(* Logix 5000 project; controller SX_V040001_C001 vendor 1 type 14 code 77 rev 16.23; software revision 16.04; part 7 of 35 *)
(* tags used below, declared in another part *)
   ALARM_BITS : INT[10];
   ALL_KINDS : INT[90];
   average_current : DINT;
   Basic : INT;
   DRIVE : INT[32];
   EMPTYING : INT[18];
   FP_ALARM_EXIST : BOOL;
   G_AInput : DINT[8];
   G_DInput : DINT[3];
   G_DOutput : DINT[3];
   loading : INT[19];
   m_alarm_exist : BOOL;
   m_alarm_horn : BOOL;
   m_notstop : BOOL;
   M_VKE_1 : BOOL;
   METERING : INT[44];
   PARAMETER : INT[501];
   pointer_dump_current : DINT;
   T_MET12_END : TIMER;
   T_MET13_END : TIMER;
   T_MET14_END : TIMER;
   T_MET_VALVE_13 : TIMER;
   T_MET_VALVE_14 : TIMER;
(* MainProgram, continued *)

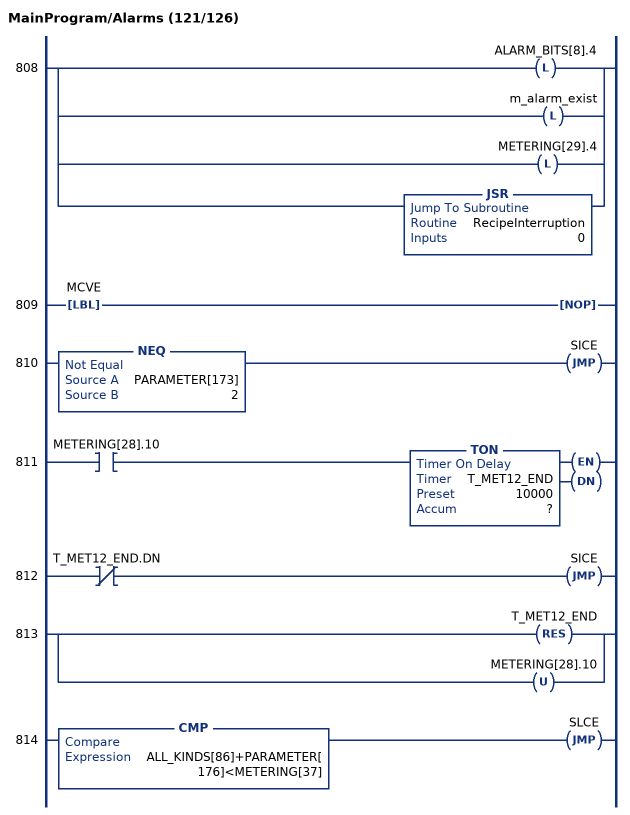
   [picture p142: MainProgram/Alarms rungs 808-814]
   808: [OTL(ALARM_BITS[8].4) ,OTL(m_alarm_exist) ,OTL(METERING[29].4) ,JSR(RecipeInterruption,0) ];
   809: LBL(MCVE)NOP();
   810: NEQ(PARAMETER[173],2)JMP(SICE);
   811: XIC(METERING[28].10)TON(T_MET12_END,?,?);
   812: XIO(T_MET12_END.DN)JMP(SICE);
   813: [RES(T_MET12_END) ,OTU(METERING[28].10) ];
   814: CMP(ALL_KINDS[86]+PARAMETER[176]<METERING[37])JMP(SLCE);
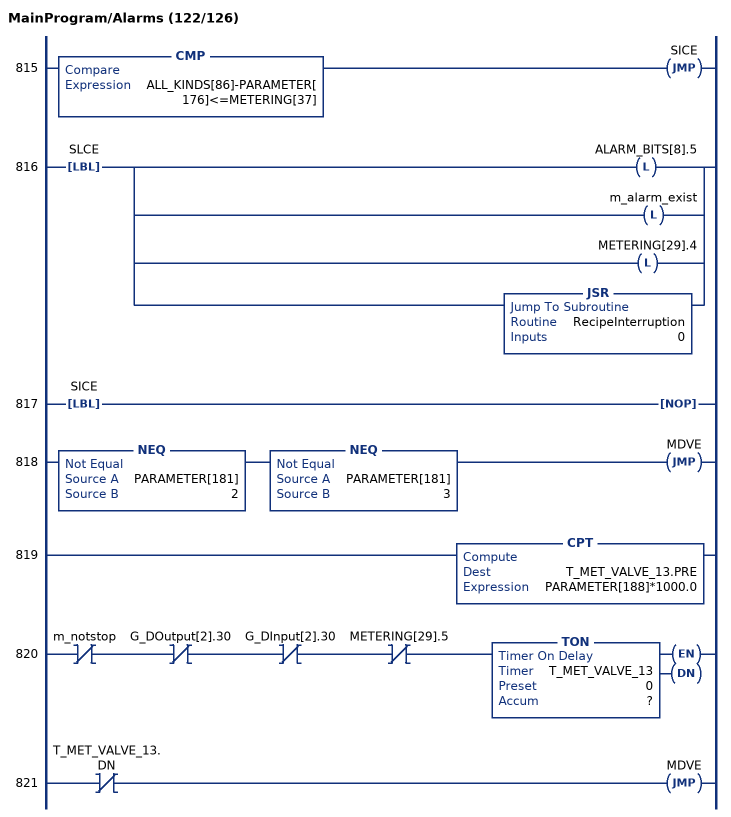
   815: CMP(ALL_KINDS[86]-PARAMETER[176]<=METERING[37])JMP(SICE);
   816: LBL(SLCE)[OTL(ALARM_BITS[8].5) ,OTL(m_alarm_exist) ,OTL(METERING[29].4) ,JSR(RecipeInterruption,0) ];
   817: LBL(SICE)NOP();
   818: NEQ(PARAMETER[181],2)NEQ(PARAMETER[181],3)JMP(MDVE);
   819: CPT(T_MET_VALVE_13.PRE,PARAMETER[188]*1000.0);
   820: XIO(m_notstop)XIO(G_DOutput[2].30)XIO(G_DInput[2].30)XIO(METERING[29].5)TON(T_MET_VALVE_13,?,?);
   821: XIO(T_MET_VALVE_13.DN)JMP(MDVE);
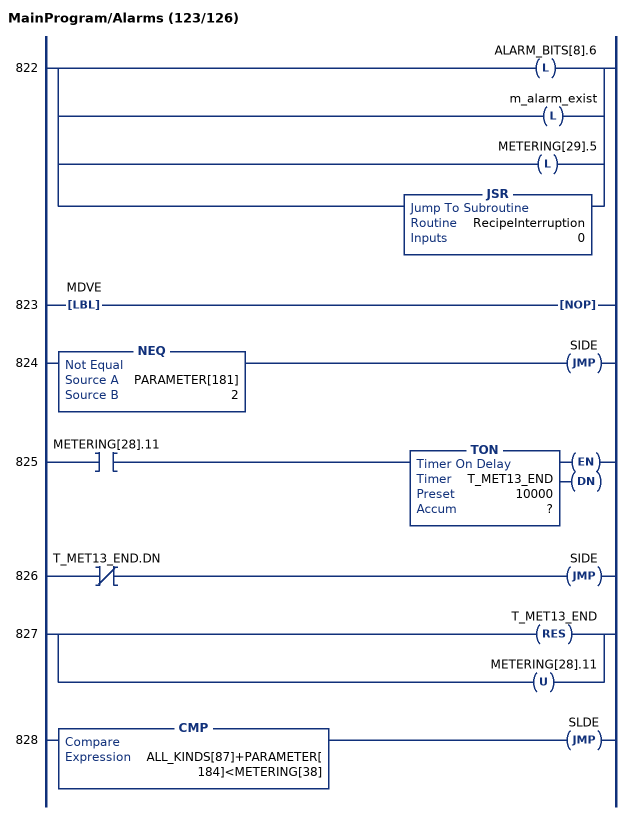
   822: [OTL(ALARM_BITS[8].6) ,OTL(m_alarm_exist) ,OTL(METERING[29].5) ,JSR(RecipeInterruption,0) ];
   823: LBL(MDVE)NOP();
   824: NEQ(PARAMETER[181],2)JMP(SIDE);
   825: XIC(METERING[28].11)TON(T_MET13_END,?,?);
   826: XIO(T_MET13_END.DN)JMP(SIDE);
   827: [RES(T_MET13_END) ,OTU(METERING[28].11) ];
   828: CMP(ALL_KINDS[87]+PARAMETER[184]<METERING[38])JMP(SLDE);
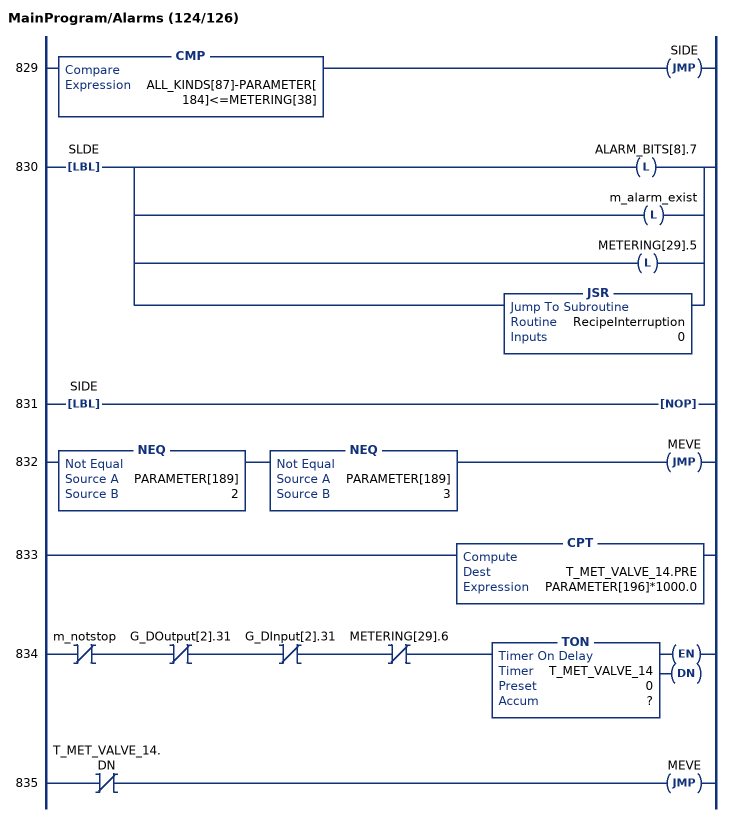
   829: CMP(ALL_KINDS[87]-PARAMETER[184]<=METERING[38])JMP(SIDE);
   830: LBL(SLDE)[OTL(ALARM_BITS[8].7) ,OTL(m_alarm_exist) ,OTL(METERING[29].5) ,JSR(RecipeInterruption,0) ];
   831: LBL(SIDE)NOP();
   832: NEQ(PARAMETER[189],2)NEQ(PARAMETER[189],3)JMP(MEVE);
   833: CPT(T_MET_VALVE_14.PRE,PARAMETER[196]*1000.0);
   834: XIO(m_notstop)XIO(G_DOutput[2].31)XIO(G_DInput[2].31)XIO(METERING[29].6)TON(T_MET_VALVE_14,?,?);
   835: XIO(T_MET_VALVE_14.DN)JMP(MEVE);
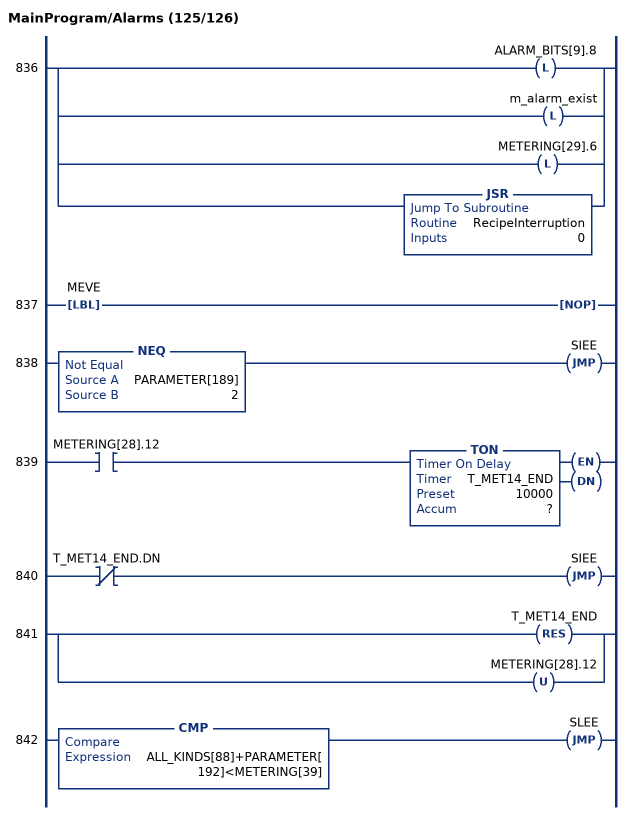
   836: [OTL(ALARM_BITS[9].8) ,OTL(m_alarm_exist) ,OTL(METERING[29].6) ,JSR(RecipeInterruption,0) ];
   837: LBL(MEVE)NOP();
   838: NEQ(PARAMETER[189],2)JMP(SIEE);
   839: XIC(METERING[28].12)TON(T_MET14_END,?,?);
   840: XIO(T_MET14_END.DN)JMP(SIEE);
   841: [RES(T_MET14_END) ,OTU(METERING[28].12) ];
   842: CMP(ALL_KINDS[88]+PARAMETER[192]<METERING[39])JMP(SLEE);
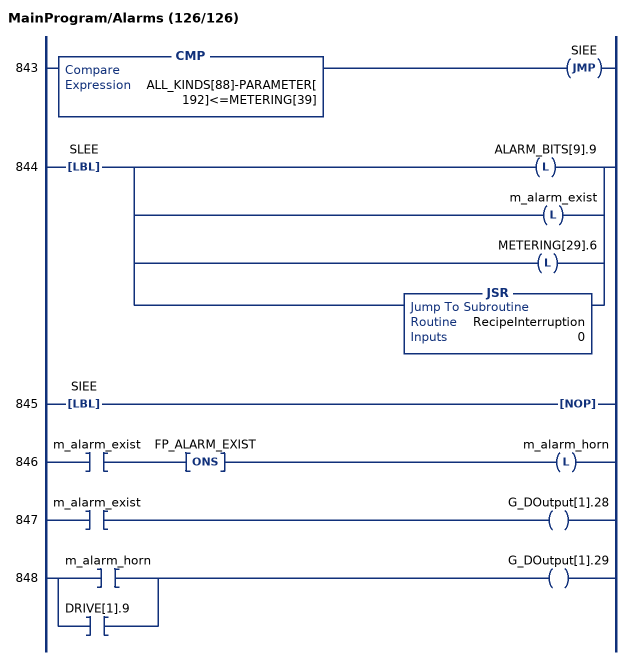
   843: CMP(ALL_KINDS[88]-PARAMETER[192]<=METERING[39])JMP(SIEE);
   844: LBL(SLEE)[OTL(ALARM_BITS[9].9) ,OTL(m_alarm_exist) ,OTL(METERING[29].6) ,JSR(RecipeInterruption,0) ];
   845: LBL(SIEE)NOP();
   846: XIC(m_alarm_exist)ONS(FP_ALARM_EXIST)OTL(m_alarm_horn);
   847: XIC(m_alarm_exist)OTE(G_DOutput[1].28);
   848: [XIC(m_alarm_horn) ,XIC(DRIVE[1].9) ]OTE(G_DOutput[1].29);
END_ROUTINE

ROUTINE aLightBeacon   (* ladder *)
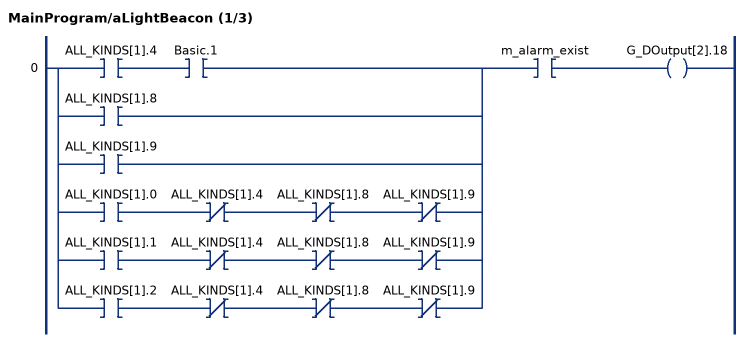
   0: [XIC(ALL_KINDS[1].4) XIC(Basic.1) ,XIC(ALL_KINDS[1].8) ,XIC(ALL_KINDS[1].9) ,XIC(ALL_KINDS[1].0) XIO(ALL_KINDS[1].4) XIO(ALL_KINDS[1].8) XIO(ALL_KINDS[1].9) ,XIC(ALL_KINDS[1].1) XIO(ALL_KINDS[1].4) XIO(ALL_KINDS[1].8) XIO(ALL_KINDS[1].9) ,XIC(ALL_KINDS[1].2) XIO(ALL_KINDS[1].4) XIO(ALL_KINDS[1].8) XIO(ALL_KINDS[1].9) ]XIC(m_alarm_exist)OTE(G_DOutput[2].18);
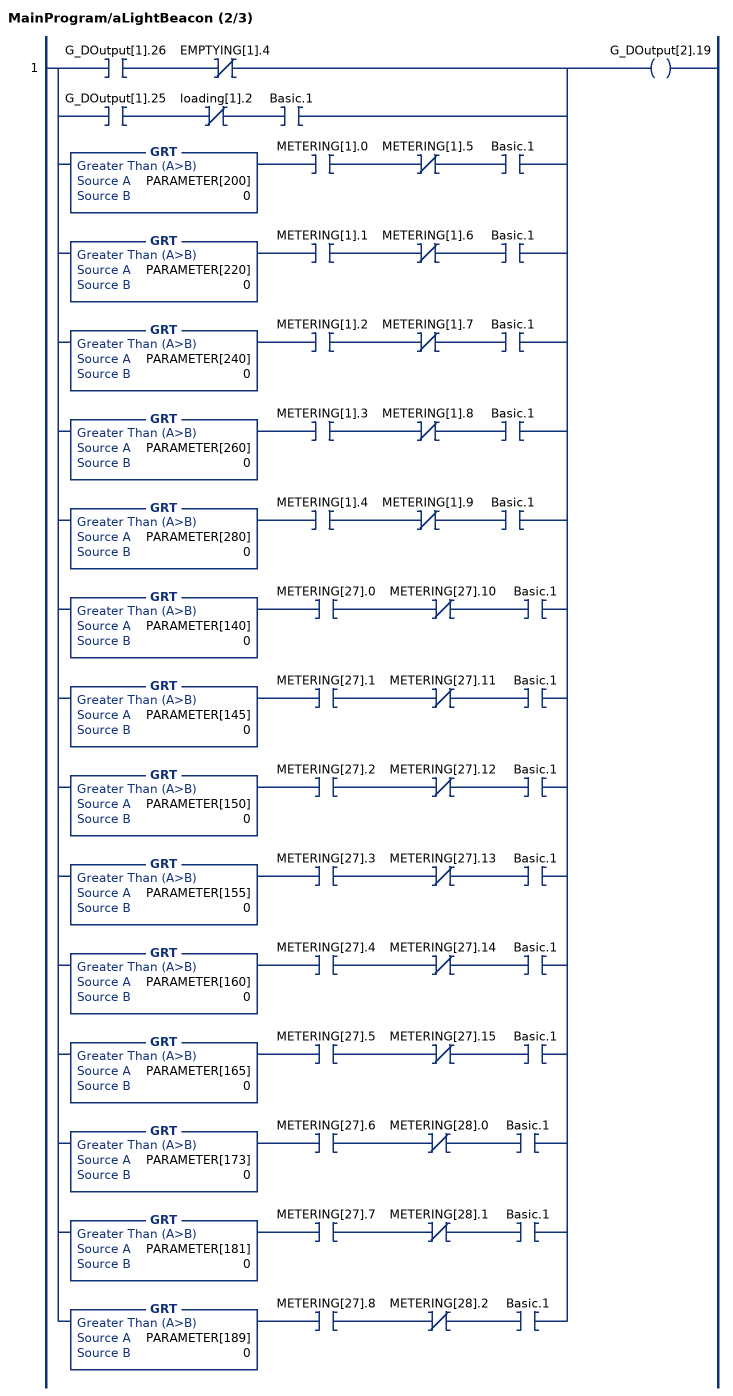
   1: [XIC(G_DOutput[1].26) XIO(EMPTYING[1].4) ,XIC(G_DOutput[1].25) XIO(loading[1].2) XIC(Basic.1) ,GRT(PARAMETER[200],0) XIC(METERING[1].0) XIO(METERING[1].5) XIC(Basic.1) ,GRT(PARAMETER[220],0) XIC(METERING[1].1) XIO(METERING[1].6) XIC(Basic.1) ,GRT(PARAMETER[240],0) XIC(METERING[1].2) XIO(METERING[1].7) XIC(Basic.1) ,GRT(PARAMETER[260],0) XIC(METERING[1].3) XIO(METERING[1].8) XIC(Basic.1) ,GRT(PARAMETER[280],0) XIC(METERING[1].4) XIO(METERING[1].9) XIC(Basic.1) ,GRT(PARAMETER[140],0) XIC(METERING[27].0) XIO(METERING[27].10) XIC(Basic.1) ,GRT(PARAMETER[145],0) XIC(METERING[27].1) XIO(METERING[27].11) XIC(Basic.1) ,GRT(PARAMETER[150],0) XIC(METERING[27].2) XIO(METERING[27].12) XIC(Basic.1) ,GRT(PARAMETER[155],0) XIC(METERING[27].3) XIO(METERING[27].13) XIC(Basic.1) ,GRT(PARAMETER[160],0) XIC(METERING[27].4) XIO(METERING[27].14) XIC(Basic.1) ,GRT(PARAMETER[165],0) XIC(METERING[27].5) XIO(METERING[27].15) XIC(Basic.1) ,GRT(PARAMETER[173],0) XIC(METERING[27].6) XIO(METERING[28].0) XIC(Basic.1) ,GRT(PARAMETER[181],0) XIC(METERING[27].7) XIO(METERING[28].1) XIC(Basic.1) ,GRT(PARAMETER[189],0) XIC(METERING[27].8) XIO(METERING[28].2) XIC(Basic.1) ]OTE(G_DOutput[2].19);
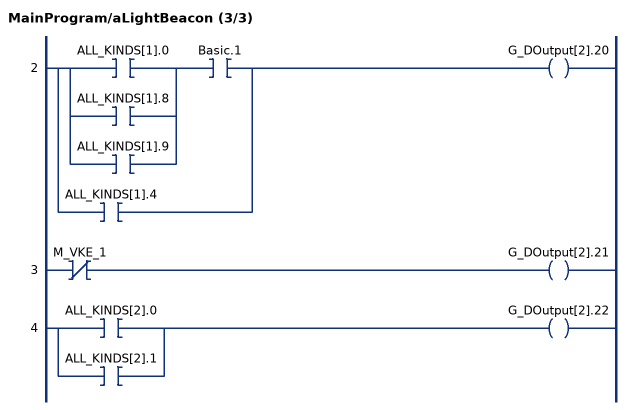
   2: [[XIC(ALL_KINDS[1].0) ,XIC(ALL_KINDS[1].8) ,XIC(ALL_KINDS[1].9) ] XIC(Basic.1) ,XIC(ALL_KINDS[1].4) ]OTE(G_DOutput[2].20);
   3: XIO(M_VKE_1)OTE(G_DOutput[2].21);
   4: [XIC(ALL_KINDS[2].0) ,XIC(ALL_KINDS[2].1) ]OTE(G_DOutput[2].22);
END_ROUTINE

ROUTINE AnalogInput   (* ladder *)
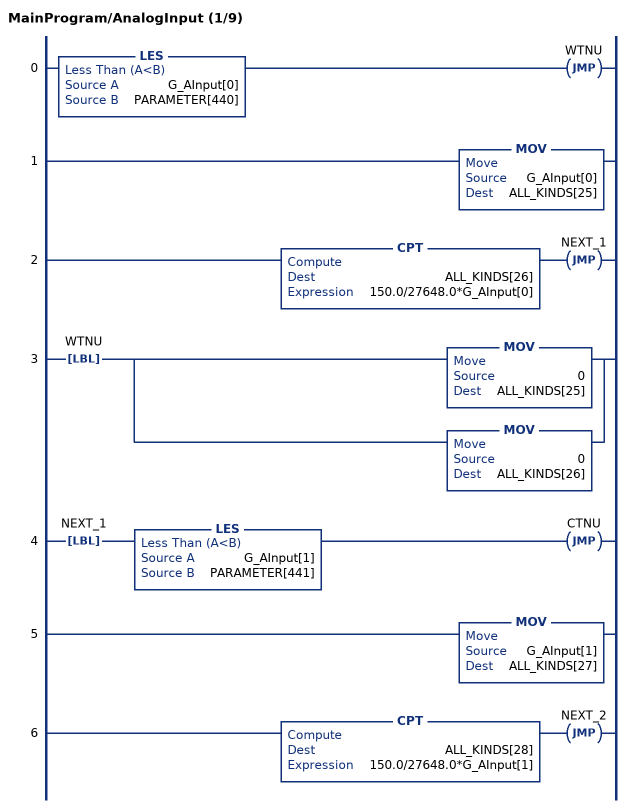
   0: LES(G_AInput[0],PARAMETER[440])JMP(WTNU);
   1: MOV(G_AInput[0],ALL_KINDS[25]);
   2: CPT(ALL_KINDS[26],150.0/27648.0*G_AInput[0])JMP(NEXT_1);
   3: LBL(WTNU)[MOV(0,ALL_KINDS[25]) ,MOV(0,ALL_KINDS[26]) ];
   4: LBL(NEXT_1)LES(G_AInput[1],PARAMETER[441])JMP(CTNU);
   5: MOV(G_AInput[1],ALL_KINDS[27]);
   6: CPT(ALL_KINDS[28],150.0/27648.0*G_AInput[1])JMP(NEXT_2);
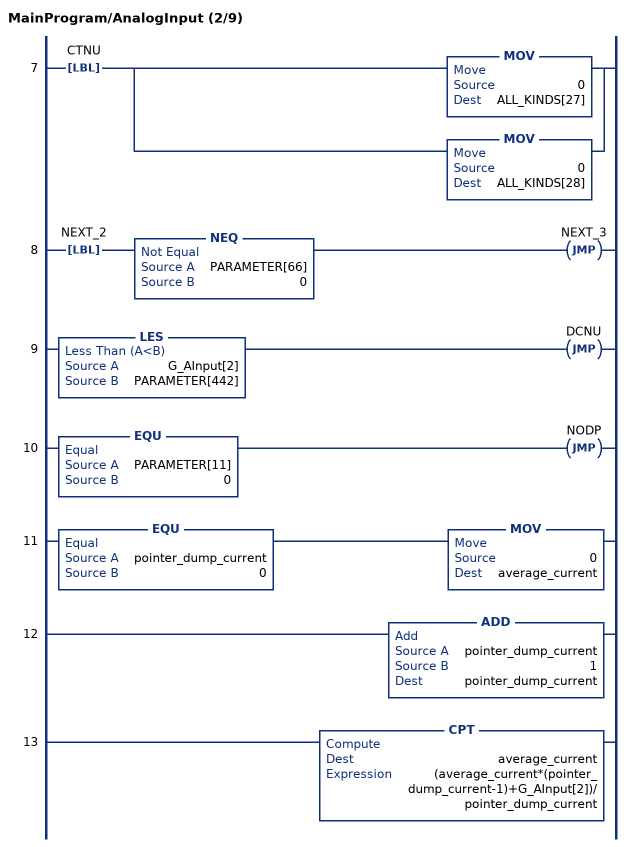
   7: LBL(CTNU)[MOV(0,ALL_KINDS[27]) ,MOV(0,ALL_KINDS[28]) ];
   8: LBL(NEXT_2)NEQ(PARAMETER[66],0)JMP(NEXT_3);
   9: LES(G_AInput[2],PARAMETER[442])JMP(DCNU);
   10: EQU(PARAMETER[11],0)JMP(NODP);
   11: EQU(pointer_dump_current,0)MOV(0,average_current);
   12: ADD(pointer_dump_current,1,pointer_dump_current);
   13: CPT(average_current,(average_current*(pointer_dump_current-1)+G_AInput[2])/pointer_dump_current);
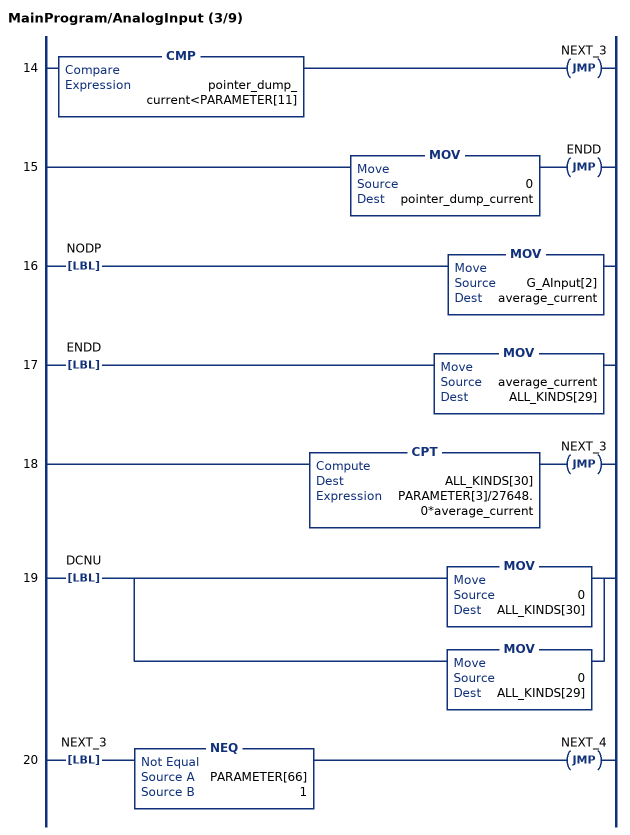
   14: CMP(pointer_dump_current<PARAMETER[11])JMP(NEXT_3);
   15: MOV(0,pointer_dump_current)JMP(ENDD);
   16: LBL(NODP)MOV(G_AInput[2],average_current);
   17: LBL(ENDD)MOV(average_current,ALL_KINDS[29]);
   18: CPT(ALL_KINDS[30],PARAMETER[3]/27648.0*average_current)JMP(NEXT_3);
   19: LBL(DCNU)[MOV(0,ALL_KINDS[30]) ,MOV(0,ALL_KINDS[29]) ];
   20: LBL(NEXT_3)NEQ(PARAMETER[66],1)JMP(NEXT_4);
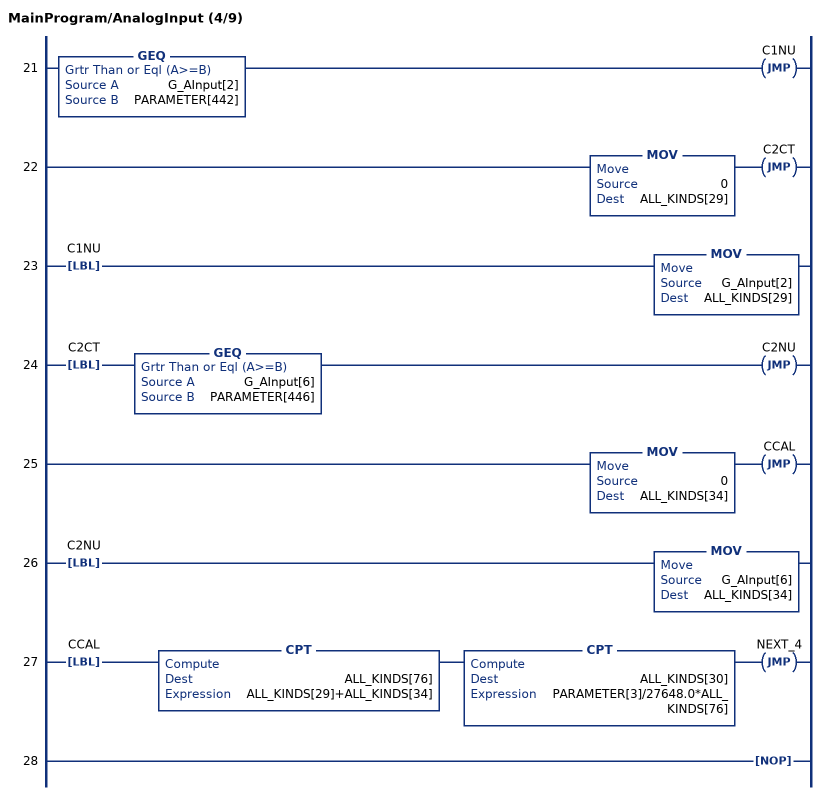
   21: GEQ(G_AInput[2],PARAMETER[442])JMP(C1NU);
   22: MOV(0,ALL_KINDS[29])JMP(C2CT);
   23: LBL(C1NU)MOV(G_AInput[2],ALL_KINDS[29]);
   24: LBL(C2CT)GEQ(G_AInput[6],PARAMETER[446])JMP(C2NU);
   25: MOV(0,ALL_KINDS[34])JMP(CCAL);
   26: LBL(C2NU)MOV(G_AInput[6],ALL_KINDS[34]);
   27: LBL(CCAL)CPT(ALL_KINDS[76],ALL_KINDS[29]+ALL_KINDS[34])CPT(ALL_KINDS[30],PARAMETER[3]/27648.0*ALL_KINDS[76])JMP(NEXT_4);
   28: NOP();
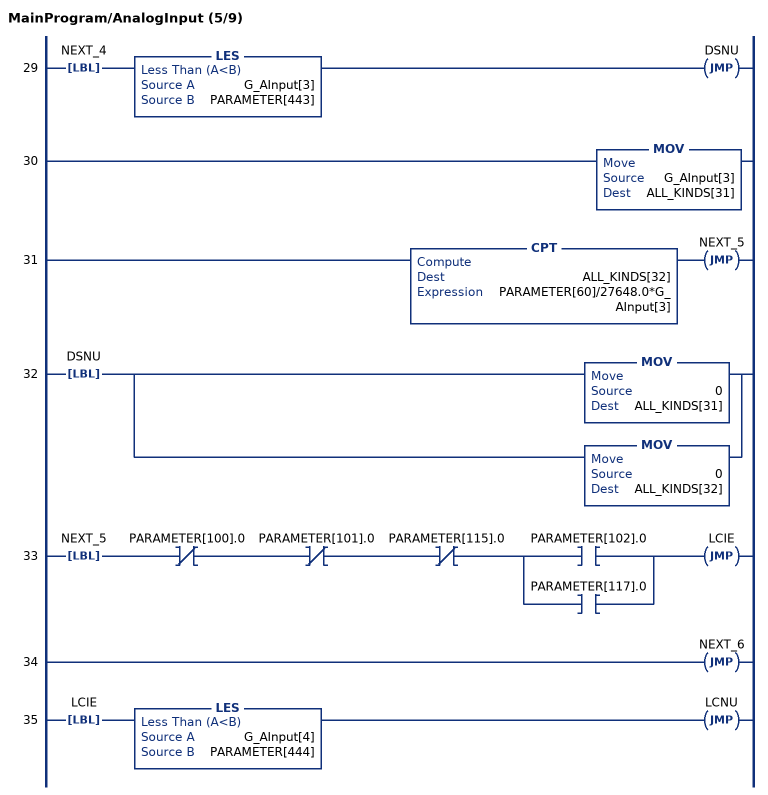
   29: LBL(NEXT_4)LES(G_AInput[3],PARAMETER[443])JMP(DSNU);
   30: MOV(G_AInput[3],ALL_KINDS[31]);
   31: CPT(ALL_KINDS[32],PARAMETER[60]/27648.0*G_AInput[3])JMP(NEXT_5);
   32: LBL(DSNU)[MOV(0,ALL_KINDS[31]) ,MOV(0,ALL_KINDS[32]) ];
   33: LBL(NEXT_5)XIO(PARAMETER[100].0)XIO(PARAMETER[101].0)XIO(PARAMETER[115].0)[XIC(PARAMETER[102].0) ,XIC(PARAMETER[117].0) ]JMP(LCIE);
   34: JMP(NEXT_6);
   35: LBL(LCIE)LES(G_AInput[4],PARAMETER[444])JMP(LCNU);
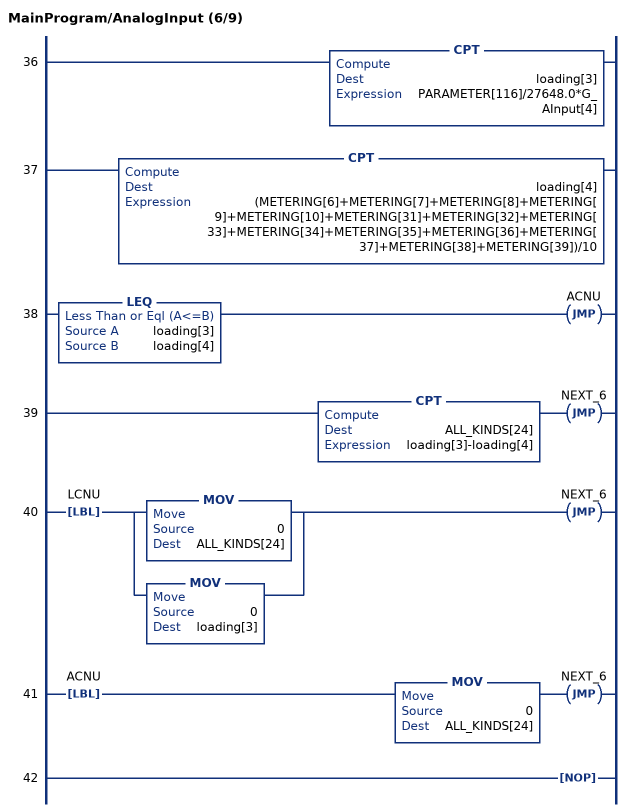
   36: CPT(loading[3],PARAMETER[116]/27648.0*G_AInput[4]);
   37: CPT(loading[4],(METERING[6]+METERING[7]+METERING[8]+METERING[9]+METERING[10]+METERING[31]+METERING[32]+METERING[33]+METERING[34]+METERING[35]+METERING[36]+METERING[37]+METERING[38]+METERING[39])/10);
   38: LEQ(loading[3],loading[4])JMP(ACNU);
   39: CPT(ALL_KINDS[24],loading[3]-loading[4])JMP(NEXT_6);
   40: LBL(LCNU)[MOV(0,ALL_KINDS[24]) ,MOV(0,loading[3]) ]JMP(NEXT_6);
   41: LBL(ACNU)MOV(0,ALL_KINDS[24])JMP(NEXT_6);
   42: NOP();
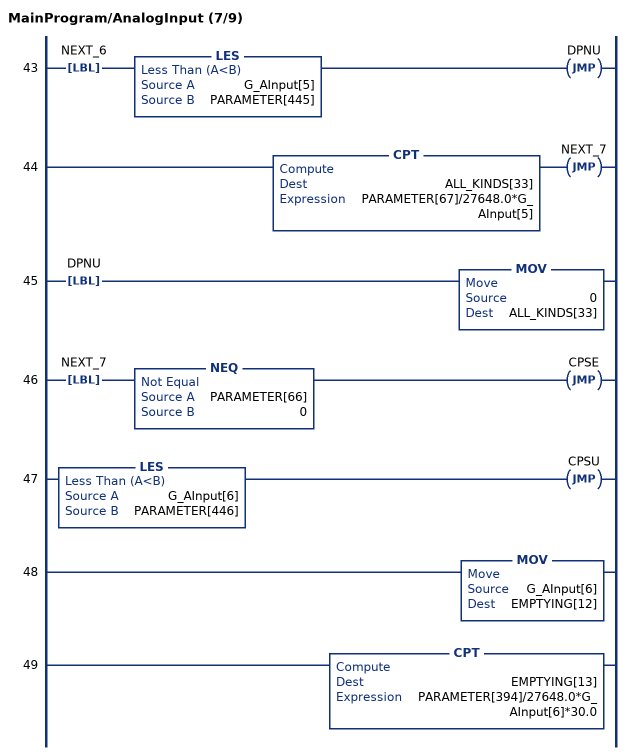
   43: LBL(NEXT_6)LES(G_AInput[5],PARAMETER[445])JMP(DPNU);
   44: CPT(ALL_KINDS[33],PARAMETER[67]/27648.0*G_AInput[5])JMP(NEXT_7);
   45: LBL(DPNU)MOV(0,ALL_KINDS[33]);
   46: LBL(NEXT_7)NEQ(PARAMETER[66],0)JMP(CPSE);
   47: LES(G_AInput[6],PARAMETER[446])JMP(CPSU);
   48: MOV(G_AInput[6],EMPTYING[12]);
   49: CPT(EMPTYING[13],PARAMETER[394]/27648.0*G_AInput[6]*30.0);
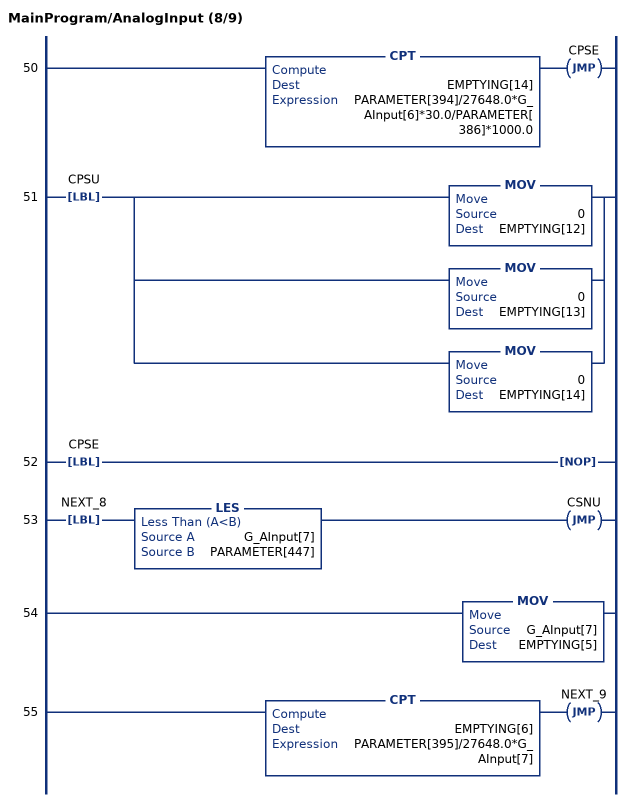
   50: CPT(EMPTYING[14],PARAMETER[394]/27648.0*G_AInput[6]*30.0/PARAMETER[386]*1000.0)JMP(CPSE);
   51: LBL(CPSU)[MOV(0,EMPTYING[12]) ,MOV(0,EMPTYING[13]) ,MOV(0,EMPTYING[14]) ];
   52: LBL(CPSE)NOP();
   53: LBL(NEXT_8)LES(G_AInput[7],PARAMETER[447])JMP(CSNU);
   54: MOV(G_AInput[7],EMPTYING[5]);
   55: CPT(EMPTYING[6],PARAMETER[395]/27648.0*G_AInput[7])JMP(NEXT_9);
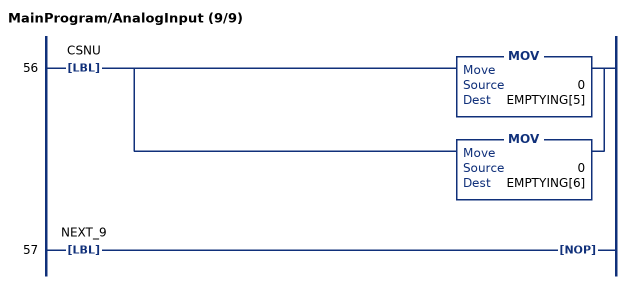
   56: LBL(CSNU)[MOV(0,EMPTYING[5]) ,MOV(0,EMPTYING[6]) ];
   57: LBL(NEXT_9)NOP();
END_ROUTINE
